// TIA Portal V17 export
// export: Created 2023-12-22T15:05:27.7974402Z, ExportSetting WithDefaults, DisplayName Totally Integrated Automation Portal, DisplayVersion V17, DisplayName TIA Portal Openness, DisplayVersion V17, DisplayName TIA Portal Version Control Interface, DisplayVersion V17, DisplayName STEP 7 Professional, DisplayVersion V17, DisplayName STEP 7 Safety, DisplayVersion V17, DisplayName WinCC Advanced, DisplayVersion V17
FUNCTION_BLOCK "DRV_Flow"   // FB130, LAD
{ S7_Optimized_Access := 'FALSE' }
VERSION : 0.1
// stored: AutoNumber false, IsIECCheckEnabled false, SetENOAutomatically false, UDAEnableTagReadback false
   VAR_IN_OUT
      impulse : Bool;
      FlowSpeed : Real;
   END_VAR
   VAR DB_SPECIFIC
      CMD : "CMD";
      Mode : Int;   // 0 - л/м, 1- л/ч, 2- м3/ч / Режим работы
      Status : Int;   // Статус устройства
      Use : Struct   // Функционал
         Indirect { S7_SetPoint := 'True'} : Bool := true;
         call_in_OB1 { S7_SetPoint := 'True'} : Bool := true;
      END_STRUCT;
      Clock { S7_SetPoint := 'True'} : Real := 0.1;   // Частота измерений
      Weight { S7_SetPoint := 'True'} : Real := 1.0;   // Вес импульса
      Time_Now : Real;
      Time_Last : Real;
      Time_Mid : Real;
      Flow_S : Real;   // литры в секунду
      Alarms : Word;   // Слово аварий
      Events : Word;   // События
      ADDR_BYTE { S7_SetPoint := 'True'} : Int;
      ADDR_BIT { S7_SetPoint := 'True'} : Int := 9;
   END_VAR
   VAR
      Filter { S7_SetPoint := 'True'} : "Filter";
   END_VAR
   VAR DB_SPECIFIC
      pos : Array[0..15] of Bool;
      Time_DTL : DTL;
   END_VAR
   VAR_TEMP
      imp : Bool;
      Filter_clock : Bool;
   END_VAR
   VAR CONSTANT
      sec : Int := 60;
   END_VAR
   // Filter.max := 100;
   VAR_TEMP   // added for the SCL form of the ladder/FBD networks
      _w1 : Bool;
      _w2 : Bool;
      _w3 : Bool;
   END_VAR
BEGIN

REGION Network 1: Чтение входа
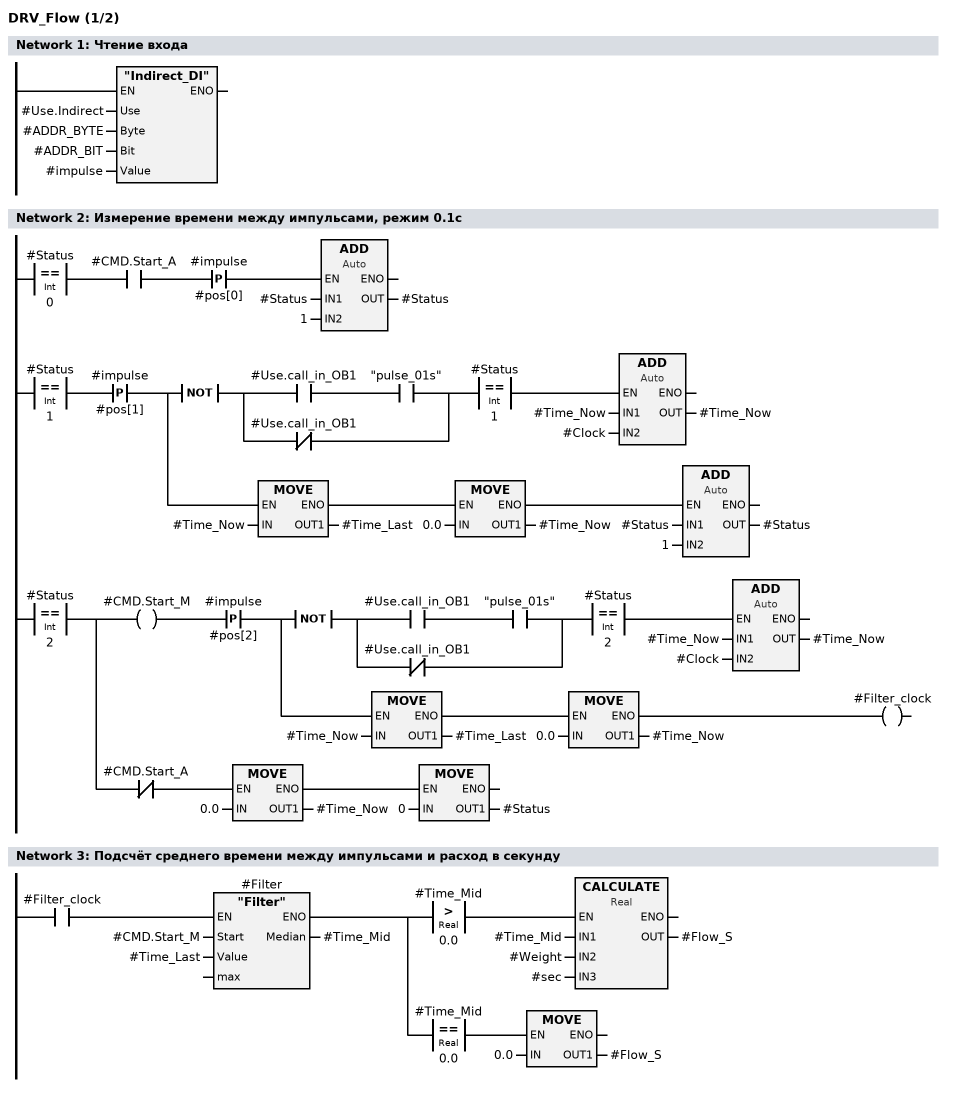
   RUNG wire#powerrail
      "Indirect_DI"(Use := #Use.Indirect, "Byte" := #ADDR_BYTE, Bit := #ADDR_BIT, Value := #impulse)
   END_RUNG
   // the same network as SCL:
   "Indirect_DI"(Use := #Use.Indirect, "Byte" := #ADDR_BYTE, Bit := #ADDR_BIT, Value := #impulse);
END_REGION

REGION Network 2: Измерение времени между импульсами, режим 0.1с
   RUNG wire#powerrail
      { S7_Templates := "SrcType := Int" } EQ_Contact(in1 := #Status, in2 := 0)
      Contact( #CMD.Start_A )
      P_Contact(operand := #impulse, bit := #pos[0])
      Add(in1 := #Status, in2 := 1, out => #Status)
   END_RUNG
   RUNG wire#powerrail
      { S7_Templates := "SrcType := Int" } EQ_Contact(in1 := #Status, in2 := 1)
      P_Contact(operand := #impulse, bit := #pos[1])
      wire#w1
      Not()
      wire#w2
      Contact( #Use.call_in_OB1 )
      Contact( "pulse_01s" )
      wire#w3
      { S7_Templates := "SrcType := Int" } EQ_Contact(in1 := #Status, in2 := 1)
      Add(in1 := #Time_Now, in2 := #Clock, out => #Time_Now)
   END_RUNG
   RUNG wire#w2
      I_Contact( #Use.call_in_OB1 )
   END_RUNG wire#w3
   RUNG wire#w1
      Move(in := #Time_Now, out1 => #Time_Last)
      Move(in := 0.0, out1 => #Time_Now)
      Add(in1 := #Status, in2 := 1, out => #Status)
   END_RUNG
   RUNG wire#powerrail
      { S7_Templates := "SrcType := Int" } EQ_Contact(in1 := #Status, in2 := 2)
      wire#w4
      Coil( #CMD.Start_M )
      P_Contact(operand := #impulse, bit := #pos[2])
      wire#w5
      Not()
      wire#w6
      Contact( #Use.call_in_OB1 )
      Contact( "pulse_01s" )
      wire#w7
      { S7_Templates := "SrcType := Int" } EQ_Contact(in1 := #Status, in2 := 2)
      Add(in1 := #Time_Now, in2 := #Clock, out => #Time_Now)
   END_RUNG
   RUNG wire#w6
      I_Contact( #Use.call_in_OB1 )
   END_RUNG wire#w7
   RUNG wire#w5
      Move(in := #Time_Now, out1 => #Time_Last)
      Move(in := 0.0, out1 => #Time_Now)
      Coil( #Filter_clock )
   END_RUNG
   RUNG wire#w4
      I_Contact( #CMD.Start_A )
      Move(in := 0.0, out1 => #Time_Now)
      Move(in := 0, out1 => #Status)
   END_RUNG
   // the same network as SCL:
   #_w1 := (#Status = 0) AND #CMD.Start_A AND #impulse AND NOT #pos[0];   // rising edge of #impulse
   #pos[0] := #impulse;
   IF #_w1 THEN #Status := #Status + 1; END_IF;
   #_w2 := (#Status = 1) AND #impulse AND NOT #pos[1];   // rising edge of #impulse
   #pos[1] := #impulse;
   IF NOT #_w2 AND ((#Use.call_in_OB1 AND "pulse_01s") OR NOT #Use.call_in_OB1) AND (#Status = 1) THEN
       #Time_Now := #Time_Now + #Clock;
   END_IF;
   IF #_w2 THEN
       #Time_Last := #Time_Now;
       #Time_Now := 0.0;
       #Status := #Status + 1;
   END_IF;
   #CMD.Start_M := #Status = 2;
   #_w3 := #CMD.Start_M AND #impulse AND NOT #pos[2];   // rising edge of #impulse
   #pos[2] := #impulse;
   IF NOT #_w3 AND ((#Use.call_in_OB1 AND "pulse_01s") OR NOT #Use.call_in_OB1) AND (#Status = 2) THEN
       #Time_Now := #Time_Now + #Clock;
   END_IF;
   IF #_w3 THEN
       #Time_Last := #Time_Now;
       #Time_Now := 0.0;
   END_IF;
   #Filter_clock := #_w3;
   IF #CMD.Start_M AND NOT #CMD.Start_A THEN
       #Time_Now := 0.0;
       #Status := 0;
   END_IF;
END_REGION

REGION Network 3: Подсчёт среднего времени между импульсами и расход в секунду
   RUNG wire#powerrail
      Contact( #Filter_clock )
      #Filter(Start := #CMD.Start_M, Value := #Time_Last, max :=, Median => #Time_Mid)
      wire#w1
      { S7_Templates := "SrcType := Real" } GT_Contact(in1 := #Time_Mid, in2 := 0.0)
      { S7_Templates := "SrcType := Real"; S7_Expression := "IN3/IN1*IN2" } Calculate(in1 := #Time_Mid, in2 := #Weight, in3 := #sec, out => #Flow_S)
   END_RUNG
   RUNG wire#w1
      { S7_Templates := "SrcType := Real" } EQ_Contact(in1 := #Time_Mid, in2 := 0.0)
      Move(in := 0.0, out1 => #Flow_S)
   END_RUNG
   // the same network as SCL:
   #Filter(EN := #Filter_clock, Start := #CMD.Start_M, Value := #Time_Last, Median => #Time_Mid, ENO => #_w1);   // "Filter"
   IF #_w1 AND (#Time_Mid > 0.0) THEN #Flow_S := #sec/#Time_Mid*#Weight; END_IF;
   IF #_w1 AND (#Time_Mid = 0.0) THEN #Flow_S := 0.0; END_IF;
END_REGION

REGION Network 4: Расход л/м, л/ч, м3/ч
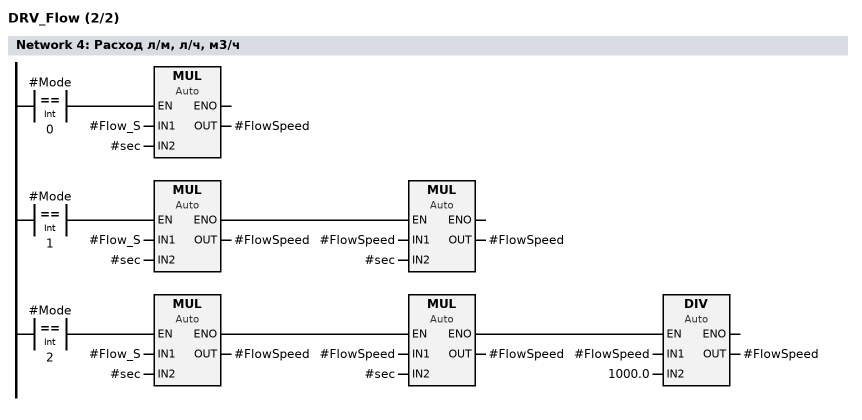
   RUNG wire#powerrail
      { S7_Templates := "SrcType := Int" } EQ_Contact(in1 := #Mode, in2 := 0)
      Mul(in1 := #Flow_S, in2 := #sec, out => #FlowSpeed)
   END_RUNG
   RUNG wire#powerrail
      { S7_Templates := "SrcType := Int" } EQ_Contact(in1 := #Mode, in2 := 1)
      Mul(in1 := #Flow_S, in2 := #sec, out => #FlowSpeed)
      Mul(in1 := #FlowSpeed, in2 := #sec, out => #FlowSpeed)
   END_RUNG
   RUNG wire#powerrail
      { S7_Templates := "SrcType := Int" } EQ_Contact(in1 := #Mode, in2 := 2)
      Mul(in1 := #Flow_S, in2 := #sec, out => #FlowSpeed)
      Mul(in1 := #FlowSpeed, in2 := #sec, out => #FlowSpeed)
      Div(in1 := #FlowSpeed, in2 := 1000.0, out => #FlowSpeed)
   END_RUNG
   // the same network as SCL:
   IF #Mode = 0 THEN #FlowSpeed := #Flow_S * #sec; END_IF;
   IF #Mode = 1 THEN
       #FlowSpeed := #Flow_S * #sec;
       #FlowSpeed := #FlowSpeed * #sec;
   END_IF;
   IF #Mode = 2 THEN
       #FlowSpeed := #Flow_S * #sec;
       #FlowSpeed := #FlowSpeed * #sec;
       #FlowSpeed := #FlowSpeed / 1000.0;
   END_IF;
END_REGION
END_FUNCTION_BLOCK
